FUNCTION_BLOCK INI_UINT (* Load and Store UDINT Data from settings.ini by Section and Key *)
  (* Standard: 61499-2; Description: based on: https://github.com/DiplomInformatikerFranzHoepfinger/SimpleIni_on_esp32 *)
  (* Version 1.0, 2022-09-23, franz *)
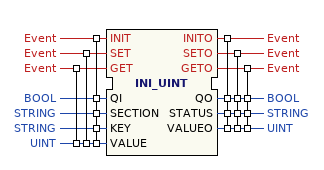
  EVENT_INPUT
    INIT WITH QI, SECTION, KEY, VALUE; (* Service Initialization *)
    SET WITH VALUE; (* set value for given key *)
    GET WITH VALUE; (* get value for given key *)
  END_EVENT
  EVENT_OUTPUT
    INITO WITH QO, STATUS, VALUEO; (* Initialization Confirm *)
    SETO WITH QO, STATUS, VALUEO; (* Confirmation of SET *)
    GETO WITH QO, STATUS, VALUEO; (* Confirmation of GET *)
  END_EVENT
  VAR_INPUT
    QI : BOOL; (* Event Input Qualifier *)
    SECTION : STRING;
    KEY : STRING; (* Key name. *)
    VALUE : UINT; (* The value to set. *)
  END_VAR
  VAR_OUTPUT
    QO : BOOL; (* Event Output Qualifier *)
    STATUS : STRING; (* Service Status *)
    VALUEO : UINT; (* The output value *)
  END_VAR
END_FUNCTION_BLOCK
